(* CODESYS project Tutorial.export
   Author: ifm electronic
   Version: 3.4.0.0
   Description: Project template for 7" ifm ecomat display 64bit device
   Title: ifm_ecomatDisplay_64bit_7Inch
   CompiledLibraryCompatibilityVersion: CODESYS V3.5 SP16 Patch 5
   Company: ifm electronic

Project tree, tasks and I/O mapping:
  Device : ecomatDisplay_64bit, ifm electronic, version 3.5.19.78
    application Application
      libraries: Standard, 3.5.18.0 (System); ifm_ecomatDisplay_Cnt, * (ifm electronic)
      task Task (cyclic, interval t#10ms, priority 1) calls PLC_PRG, P_VehicleSpeed, P_DateTime, P_Main
      task VISU_TASK (cyclic, interval t#20ms, priority 15) calls VisuElems.Visu_Prg
      GlobalVariables/
        Enums/
          global variables ScreenIDs
        global variables GLV_MVC
        global variables GVL_KeyList
        global variables GVL_KeyList_FT
        global variables GVL_KeyList_RT
      MVC/
        Controller/
          MainScreen/
            function block FB_MainScreen [ST]
          Profiles/
          Settings/
            function block FB_Settings [ST]
          function block FB_Router [ST]
        Model/
          program P_DateTime [ST]
          program P_VehicleSpeed [ST]
        View/
          Settings/
            Widgets/
              visualisation Angle
              visualisation Graph
            visualisation Settings
          visualisation Background
          visualisation MainScreen
          visualisation Profiles
      TextLists/
        text list TL_eKeyMapCodes
      image pool ifmImagePool
      program PLC_PRG [FBD]: ACT_KeyList_FT, ACT_KeyList_RT
      program PLC_PRG_IN_ST [ST]: ACT_KeyList_FT, ACT_KeyList_RT
      program P_Main [ST]
    Communication : Communication, ifm electronic, version 3.5.19.78
      Ethernet : Ethernet, ifm electronic, version 3.5.19.78
      CAN : CAN, ifm electronic, version 3.5.19.78
        CANbus : CANbus, ifm electronic, version 3.0.0.0
          J1939_Manager : J1939_Manager, CODESYS, version 4.2.0.0
            RX_Tutorial : J1939_ECU, CODESYS, version 4.2.0.0
                settings: NAME = 16#0000000000000000; Communication Watchdog Timeout Period = 16#05DC ms; Activated PGs = 1; PG Offline Data.Name = "My_PGN"; PG Offline Data.Description = ""; PG Online Data.PGN = 65285; PG Online Data.Length (Bytes) = 8; PG Transmission Settings.Destination Address = 255; PG Transmission Settings.CycleTimeFactor = 1; Signal Offline Data.SPN = 1; Signal Offline Data.Name = "RX_Speed"; Signal Offline Data.Description = ""; Signal Offline Data.Unit = ""; Signal Offline Data.Min = 0; Signal Offline Data.Max = 0; Signal Online Data.BitSize = 8; Signal Online Data.BitPosition = 0; Convert Data.Flags = 3; Convert Data.pSigValue = 0; Convert Data.Scaling = 4607182418800017408; Convert Data.Offset = 0
                input  RX_Speed : USINT  // RX_Speed
            TX_Motor : J1939_ECU, CODESYS, version 4.2.0.0
                settings: NAME = 16#0000000000000000; Local Device = TRUE; Communication Watchdog Timeout Period = 16#05DC ms; Activated PGs = 1; PG Offline Data.Name = "TX_Speed"; PG Offline Data.Description = ""; PG Online Data.PGN = 65286; PG Online Data.Length (Bytes) = 8; PG Transmission Settings.Destination Address = 255; PG Transmission Settings.CycleTimeFactor = 5; Signal Offline Data.SPN = 0; Signal Offline Data.Name = "TX_ModifiedSpeed"; Signal Offline Data.Description = ""; Signal Offline Data.Unit = ""; Signal Offline Data.Min = 0; Signal Offline Data.Max = 0; Signal Online Data.BitSize = 8; Signal Online Data.BitPosition = 0; Convert Data.Flags = 3; Convert Data.pSigValue = 0; Convert Data.Scaling = 4607182418800017408; Convert Data.Offset = 0; Activated PGs = 0
                output Application.P_VehicleSpeed.uSpeed : USINT  // TX_ModifiedSpeed
  Project Information/
  text list GlobalTextList
  text list System
  5ce3da45-db07-42e7-a21c-a00fff4ed8f6|E:\BSR\Me\May Be Useful\ifm-engg_Logo\IFMLO_PANT_2c.png
  5ce3da45-db07-42e7-a21c-a00fff4ed8f6|E:\BSR\OnSVN\CODESYS_V3x\PDM360-3\DesignDocs\Pictures\7Inch\Bg_7Inch_dark.png
  5ce3da45-db07-42e7-a21c-a00fff4ed8f6|E:\BSR\OnSVN\CODESYS_V3x\PDM360-3\DesignDocs\Pictures\7Inch\Bg_7Inch_light.png
  5ce3da45-db07-42e7-a21c-a00fff4ed8f6|E:\BSR\OnSVN\CODESYS_V3x\PDM360-3\DesignDocs\Pictures\7Inch\Button_7Inch_dark.png
  5ce3da45-db07-42e7-a21c-a00fff4ed8f6|E:\BSR\OnSVN\CODESYS_V3x\PDM360-3\DesignDocs\Pictures\7Inch\Button_7Inch_light.png
  5ce3da45-db07-42e7-a21c-a00fff4ed8f6|E:\BSR\OnSVN\CODESYS_V3x\PDM360-3\DesignDocs\Pictures\7Inch\Button_And_Bg_7Inch_dark.png
  5ce3da45-db07-42e7-a21c-a00fff4ed8f6|E:\BSR\OnSVN\CODESYS_V3x\PDM360-3\DesignDocs\Pictures\7Inch\Button_And_Bg_7Inch_light.png
*)

// Device/Application/GlobalVariables/GLV_MVC

VAR_GLOBAL
	ScreenID : eScreenID := eScreenID.Main;
END_VAR

// Device/Application/GlobalVariables/GVL_KeyList
{attribute 'qualified_only'}

(* 

!!! This GVL list is from project template !!!

The following variables are controlled by key events mapped at Default Hotkey mapping list in Visualization Manager.

For example, F1 function key of standard keyboard (MFII) is pressed, xF1 bit in this list will become TRUE; when the same 
key is released then xF1 become FALSE.

*)

VAR_GLOBAL

(* Display system key press / release event status. TRUE = Key Pressed, FALSE = Key Released  *)
	xF1 		: BOOL;		(* Event status of F1 function key *)
	xF2 		: BOOL;		(* Event status of F2 function key *)
	xF3 		: BOOL;		(* Event status of F3 function key *)
	xF4 		: BOOL;		(* Event status of F4 function key *)
	xF5 		: BOOL;		(* Event status of F5 function key *)
	xF6 		: BOOL;		(* Event status of F6 function key *)
	xF7 		: BOOL;		(* Event status of F7 function key *)
	xF8 		: BOOL;		(* Event status of F8 function key *)
	xF9 		: BOOL;		(* Event status of F9 function key *)
	xF10 		: BOOL;		(* Event status of F10 function key *)
	xUp 		: BOOL;		(* Event status of Up arrow key *)
	xDown		: BOOL;		(* Event status of Down arrow key *)
	xLeft 		: BOOL;		(* Event status of Left arrow key *)
	xRight 		: BOOL;		(* Event status of Right arrow key *)
	xKey_Return : BOOL;		(* Event status of Return (or Enter) key *)
END_VAR

// Device/Application/GlobalVariables/GVL_KeyList_FT
{attribute 'qualified_only'}

(* 

!!! This GVL list is from project template !!!

The following variables returns a pulse for one scan cycle when a respective key is released (i.e. at falling trigger).
These key release event is detected by the state of variables in GVL GVL_KeyList.

For example, F1 function key of standard keyboard (MFII) is released, xF1 bit in this list will become TRUE for one scan cycle.

*)

VAR_GLOBAL

(* Display system key release event falling trigger pulse. *)
	xF1 		: BOOL;		(* Event status of F1 function key *)
	xF2 		: BOOL;		(* Event status of F2 function key *)
	xF3 		: BOOL;		(* Event status of F3 function key *)
	xF4 		: BOOL;		(* Event status of F4 function key *)
	xF5 		: BOOL;		(* Event status of F5 function key *)
	xF6 		: BOOL;		(* Event status of F6 function key *)
	xF7 		: BOOL;		(* Event status of F7 function key *)
	xF8 		: BOOL;		(* Event status of F8 function key *)
	xF9 		: BOOL;		(* Event status of F9 function key *)
	xF10 		: BOOL;		(* Event status of F10 function key *)
	xUp 		: BOOL;		(* Event status of Up arrow key *)
	xDown		: BOOL;		(* Event status of Down arrow key *)
	xLeft 		: BOOL;		(* Event status of Left arrow key *)
	xRight 		: BOOL;		(* Event status of Right arrow key *)
	xKey_Return : BOOL;		(* Event status of Return (or Enter) key *)
END_VAR

// Device/Application/GlobalVariables/GVL_KeyList_RT
{attribute 'qualified_only'}

(* 

!!! This GVL list is from project template !!!

The following variables returns a pulse for one scan cycle when a respective key is pressed (i.e. at rising trigger)
These key press event is detected by the state of variables in GVL GVL_KeyList.

For example, F1 function key of standard keyboard (MFII) is pressed, xF1 bit in this list will become TRUE for one scan cycle.

*)

VAR_GLOBAL

(*Display system key press event rising trigger pulse *)
	xF1 		: BOOL;		(* Event status of F1 function key *)
	xF2 		: BOOL;		(* Event status of F2 function key *)
	xF3 		: BOOL;		(* Event status of F3 function key *)
	xF4 		: BOOL;		(* Event status of F4 function key *)
	xF5 		: BOOL;		(* Event status of F5 function key *)
	xF6 		: BOOL;		(* Event status of F6 function key *)
	xF7 		: BOOL;		(* Event status of F7 function key *)
	xF8 		: BOOL;		(* Event status of F8 function key *)
	xF9 		: BOOL;		(* Event status of F9 function key *)
	xF10 		: BOOL;		(* Event status of F10 function key *)
	xUp 		: BOOL;		(* Event status of Up arrow key *)
	xDown		: BOOL;		(* Event status of Down arrow key *)
	xLeft 		: BOOL;		(* Event status of Left arrow key *)
	xRight 		: BOOL;		(* Event status of Right arrow key *)
	xKey_Return : BOOL;		(* Event status of Return (or Enter) key *)
END_VAR

// Device/Application/GlobalVariables/Enums/ScreenIDs
{attribute 'qualified_only'}
VAR_GLOBAL
END_VAR

TYPE eScreenID : (
  Main := 0,
  Settings := 1
);
END_TYPE

// Device/Application/PLC_PRG

(* !!! This POU is from project template !!! *)

PROGRAM PLC_PRG
VAR
(* Below is the FB instance with initial values to set default key mapping. The default key map is as per the default values set for ifmDevice.stKEY_MAP_LIST. *)
	fbSetKeyMapping		: ifmDevice.SetKeyMapping;

(* Below is the FB instance with initial values to hide splash screen and show CODESYS visualisation if a visualization exists in the application. In this case 
Visu_Default is displayed. *)
	fbHideSplashScreen	: ifmDevice.HideSplashScreen;

END_VAR
VAR // added by the converter: edge detectors and wires of the graphical bodies
    _ft1, _ft2, _ft3, _ft4, _ft5, _ft6, _ft7, _ft8, _ft9, _ft10, _ft11, _ft12, _ft13, _ft14, _ft15 : F_TRIG;
    _rt1, _rt2, _rt3, _rt4, _rt5, _rt6, _rt7, _rt8, _rt9, _rt10, _rt11, _rt12, _rt13, _rt14, _rt15 : R_TRIG;
END_VAR

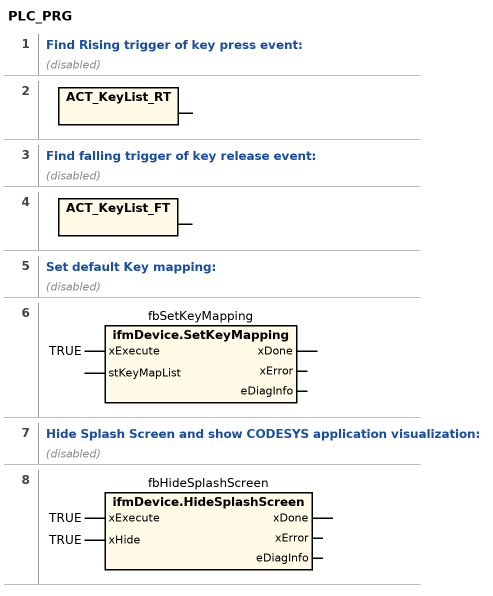
// NETWORK 1 (disabled)
// label: Find Rising trigger of key press event

// NETWORK 2
ACT_KeyList_RT();

// NETWORK 3 (disabled)
// label: Find falling trigger of key release event

// NETWORK 4
ACT_KeyList_FT();

// NETWORK 5 (disabled)
// label: Set default Key mapping

// NETWORK 6
fbSetKeyMapping(xExecute := TRUE); // ifmDevice.SetKeyMapping

// NETWORK 7 (disabled)
// label: Hide Splash Screen and show CODESYS application visualization

// NETWORK 8
fbHideSplashScreen(xExecute := TRUE, xHide := TRUE); // ifmDevice.HideSplashScreen

ACTION ACT_KeyList_FT:
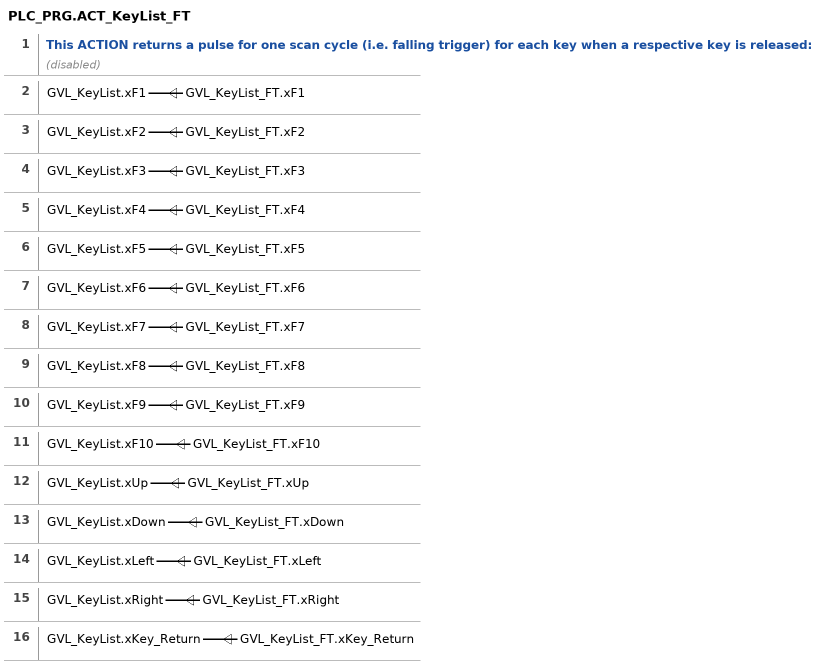
// NETWORK 1 (disabled)
// label: This ACTION returns a pulse for one scan cycle (i.e. falling trigger) for each key when a respective key is released

// NETWORK 2
_ft1(CLK := GVL_KeyList.xF1);
GVL_KeyList_FT.xF1 := _ft1.Q;

// NETWORK 3
_ft2(CLK := GVL_KeyList.xF2);
GVL_KeyList_FT.xF2 := _ft2.Q;

// NETWORK 4
_ft3(CLK := GVL_KeyList.xF3);
GVL_KeyList_FT.xF3 := _ft3.Q;

// NETWORK 5
_ft4(CLK := GVL_KeyList.xF4);
GVL_KeyList_FT.xF4 := _ft4.Q;

// NETWORK 6
_ft5(CLK := GVL_KeyList.xF5);
GVL_KeyList_FT.xF5 := _ft5.Q;

// NETWORK 7
_ft6(CLK := GVL_KeyList.xF6);
GVL_KeyList_FT.xF6 := _ft6.Q;

// NETWORK 8
_ft7(CLK := GVL_KeyList.xF7);
GVL_KeyList_FT.xF7 := _ft7.Q;

// NETWORK 9
_ft8(CLK := GVL_KeyList.xF8);
GVL_KeyList_FT.xF8 := _ft8.Q;

// NETWORK 10
_ft9(CLK := GVL_KeyList.xF9);
GVL_KeyList_FT.xF9 := _ft9.Q;

// NETWORK 11
_ft10(CLK := GVL_KeyList.xF10);
GVL_KeyList_FT.xF10 := _ft10.Q;

// NETWORK 12
_ft11(CLK := GVL_KeyList.xUp);
GVL_KeyList_FT.xUp := _ft11.Q;

// NETWORK 13
_ft12(CLK := GVL_KeyList.xDown);
GVL_KeyList_FT.xDown := _ft12.Q;

// NETWORK 14
_ft13(CLK := GVL_KeyList.xLeft);
GVL_KeyList_FT.xLeft := _ft13.Q;

// NETWORK 15
_ft14(CLK := GVL_KeyList.xRight);
GVL_KeyList_FT.xRight := _ft14.Q;

// NETWORK 16
_ft15(CLK := GVL_KeyList.xKey_Return);
GVL_KeyList_FT.xKey_Return := _ft15.Q;
END_ACTION

ACTION ACT_KeyList_RT:
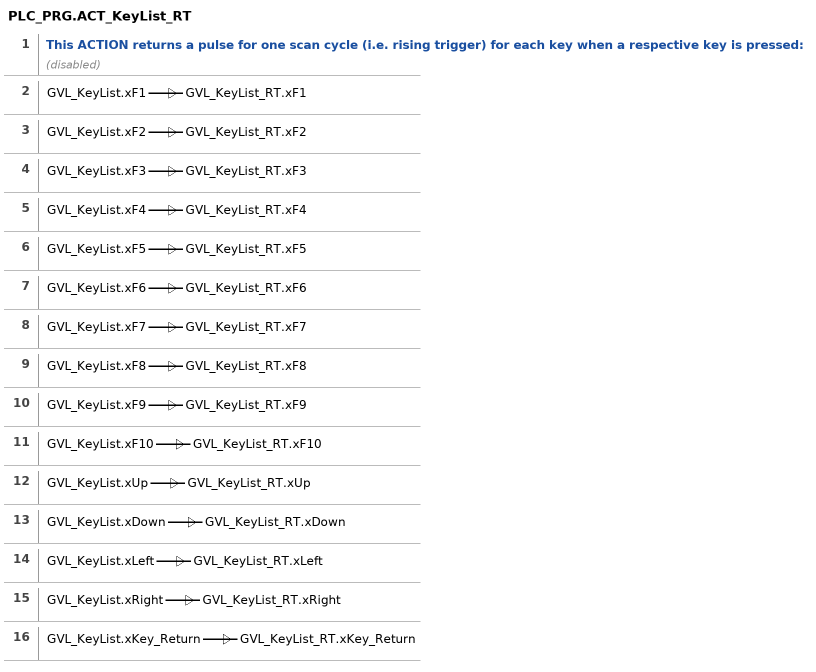
// NETWORK 1 (disabled)
// label: This ACTION returns a pulse for one scan cycle (i.e. rising trigger) for each key when a respective key is pressed

// NETWORK 2
_rt1(CLK := GVL_KeyList.xF1);
GVL_KeyList_RT.xF1 := _rt1.Q;

// NETWORK 3
_rt2(CLK := GVL_KeyList.xF2);
GVL_KeyList_RT.xF2 := _rt2.Q;

// NETWORK 4
_rt3(CLK := GVL_KeyList.xF3);
GVL_KeyList_RT.xF3 := _rt3.Q;

// NETWORK 5
_rt4(CLK := GVL_KeyList.xF4);
GVL_KeyList_RT.xF4 := _rt4.Q;

// NETWORK 6
_rt5(CLK := GVL_KeyList.xF5);
GVL_KeyList_RT.xF5 := _rt5.Q;

// NETWORK 7
_rt6(CLK := GVL_KeyList.xF6);
GVL_KeyList_RT.xF6 := _rt6.Q;

// NETWORK 8
_rt7(CLK := GVL_KeyList.xF7);
GVL_KeyList_RT.xF7 := _rt7.Q;

// NETWORK 9
_rt8(CLK := GVL_KeyList.xF8);
GVL_KeyList_RT.xF8 := _rt8.Q;

// NETWORK 10
_rt9(CLK := GVL_KeyList.xF9);
GVL_KeyList_RT.xF9 := _rt9.Q;

// NETWORK 11
_rt10(CLK := GVL_KeyList.xF10);
GVL_KeyList_RT.xF10 := _rt10.Q;

// NETWORK 12
_rt11(CLK := GVL_KeyList.xUp);
GVL_KeyList_RT.xUp := _rt11.Q;

// NETWORK 13
_rt12(CLK := GVL_KeyList.xDown);
GVL_KeyList_RT.xDown := _rt12.Q;

// NETWORK 14
_rt13(CLK := GVL_KeyList.xLeft);
GVL_KeyList_RT.xLeft := _rt13.Q;

// NETWORK 15
_rt14(CLK := GVL_KeyList.xRight);
GVL_KeyList_RT.xRight := _rt14.Q;

// NETWORK 16
_rt15(CLK := GVL_KeyList.xKey_Return);
GVL_KeyList_RT.xKey_Return := _rt15.Q;
END_ACTION

END_PROGRAM

// Device/Application/MVC/Model/P_VehicleSpeed
PROGRAM P_VehicleSpeed
VAR
	// currently requested speed
	uPercentage : USINT :=  0;
	
	// upper speed barier in km/h
	UPPER_SPEED_BARRIER : USINT := 190;
	
	// speed output for the motor
	uSpeed : USINT := 0;
END_VAR


// calculate our percentage from CAN input
uPercentage := RX_Speed * 10; 

// calculate the speed:  1% = 2km/h
IF (UPPER_SPEED_BARRIER < uPercentage * 2) THEN 	// check if the pedal is floored
	uSpeed := UPPER_SPEED_BARRIER; 					// if yes, allow only 95% of possible speed
	ELSE
	uSpeed := uPercentage * 2;					// else, use the calculated value
	
	
END_IF

END_PROGRAM

// Device/Application/MVC/Model/P_DateTime
PROGRAM P_DateTime
VAR
	GetSysTimeCyclic :ifmDevice.GetSysTime;
	DateTime :ifmDevice.stDATE_TIME;
END_VAR

GetSysTimeCyclic(
	xExecute:= TRUE , 
	xDone=> , 
	xError=> , 
	eDiagInfo=> , 
	stDateTime=> DateTime , 
	sTimeZone=> , 
	xNTP_DateTime=> );

END_PROGRAM

// Device/Application/P_Main
PROGRAM P_Main
VAR
	FB_Router : FB_Router;
END_VAR

FB_Router();

END_PROGRAM

// Device/Application/MVC/Controller/FB_Router
FUNCTION_BLOCK FB_Router
VAR_INPUT
END_VAR
VAR_OUTPUT
END_VAR
VAR
	FB_MainScreen : FB_MainScreen;
	FB_Settings : FB_Settings;
END_VAR




case ScreenID OF
		Main : FB_MainScreen();
		Settings : FB_Settings();
END_CASE

END_FUNCTION_BLOCK

// Device/Application/MVC/Controller/MainScreen/FB_MainScreen
FUNCTION_BLOCK FB_MainScreen
VAR_INPUT
END_VAR
VAR_OUTPUT
END_VAR
VAR
	uTest: udint := 0;
END_VAR

IF GVL_KeyList_FT.xF3 THEN
	ScreenID := 1;
END_IF

END_FUNCTION_BLOCK

// Device/Application/MVC/Controller/Settings/FB_Settings
FUNCTION_BLOCK FB_Settings
VAR_INPUT
END_VAR
VAR_OUTPUT
END_VAR
VAR
	MAX_WIDGET_INDEX :SINT := 1;
	// active widget index
	sWidgetIndex : SINT := 0;
END_VAR


// go back to HOME
IF GVL_KeyList_FT.xF5 THEN
	ScreenID := 0;
END_IF



// switch wigdet to left
IF GVL_KeyList_FT.xLeft THEN
    sWidgetIndex := (sWidgetIndex - 1 + MAX_WIDGET_INDEX + 1) MOD (MAX_WIDGET_INDEX + 1);
END_IF

// switch wigdet to right
IF GVL_KeyList_FT.xRight THEN
    sWidgetIndex := (sWidgetIndex + 1) MOD (MAX_WIDGET_INDEX + 1);
END_IF

END_FUNCTION_BLOCK

// Device/Application/PLC_PRG_IN_ST

(* !!! This POU is from project template !!! *)

PROGRAM PLC_PRG_IN_ST
VAR
(* Below is the FB instance with initial values to set default key mapping. The default key map is as per the default values set for ifmDevice.stKEY_MAP_LIST *)
	fbSetKeyMapping		: ifmDevice.SetKeyMapping;

(* Below is the FB instance with initial values to hide splash screen and show CODESYS visualisation if a visualization exists in the application. In this case 
Visu_Default is displayed. *)
	fbHideSplashScreen	: ifmDevice.HideSplashScreen;

(* Find rising trigger of key press event *)
	fbRTrig		: ARRAY[0..14] OF Standard.R_TRIG;
 
(* Find falling trigger of key release event *)
	fbFTrig		: ARRAY[0..14] OF Standard.F_TRIG; 
END_VAR

(* Find rising trigger of key press event *)
ACT_KeyList_RT();

(* Find falling trigger of key release event *)
ACT_KeyList_FT();


(* Set default key mapping *)
fbSetKeyMapping(
	xExecute		:= TRUE,
	stKeyMapList	:= , 
	xDone			=> , 
	xError			=> , 
	eDiagInfo		=> );

(* Hide splash screen and show CODESYS application visualization *)
fbHideSplashScreen(
	xExecute	:= TRUE,
	xHide		:= TRUE,
	xDone		=> , 
	xError		=> , 
	eDiagInfo	=> );

ACTION ACT_KeyList_FT:

(* This ACTION returns a pulse for one scan cycle (i.e. falling trigger) for each key when a respective key is released *)

fbFTrig[0](CLK := GVL_KeyList.xF1, 		Q => GVL_KeyList_FT.xF1);
fbFTrig[1](CLK := GVL_KeyList.xF2, 		Q => GVL_KeyList_FT.xF2);
fbFTrig[2](CLK := GVL_KeyList.xF3, 		Q => GVL_KeyList_FT.xF3);
fbFTrig[3](CLK := GVL_KeyList.xF4, 		Q => GVL_KeyList_FT.xF4);
fbFTrig[4](CLK := GVL_KeyList.xF5, 		Q => GVL_KeyList_FT.xF5);
fbFTrig[5](CLK := GVL_KeyList.xF6, 		Q => GVL_KeyList_FT.xF6);
fbFTrig[6](CLK := GVL_KeyList.xF7, 		Q => GVL_KeyList_FT.xF7);
fbFTrig[7](CLK := GVL_KeyList.xF8,		Q => GVL_KeyList_FT.xF8);
fbFTrig[8](CLK := GVL_KeyList.xF9, 		Q => GVL_KeyList_FT.xF9);
fbFTrig[9](CLK := GVL_KeyList.xF10, 	Q => GVL_KeyList_FT.xF10);

fbFTrig[10](CLK := GVL_KeyList.xUp, 	Q => GVL_KeyList_FT.xUp);
fbFTrig[11](CLK := GVL_KeyList.xDown,	Q => GVL_KeyList_FT.xDown);
fbFTrig[12](CLK := GVL_KeyList.xLeft,	Q => GVL_KeyList_FT.xLeft);
fbFTrig[13](CLK := GVL_KeyList.xRight,	Q => GVL_KeyList_FT.xRight);
fbFTrig[14](CLK := GVL_KeyList.xKey_Return, Q => GVL_KeyList_FT.xKey_Return);
END_ACTION

ACTION ACT_KeyList_RT:

(* This ACTION returns a pulse for one scan cycle (i.e. rising trigger) for each key when a respective key is pressed *)
fbRTrig[0](CLK := GVL_KeyList.xF1, 		Q => GVL_KeyList_RT.xF1);
fbRTrig[1](CLK := GVL_KeyList.xF2, 		Q => GVL_KeyList_RT.xF2);
fbRTrig[2](CLK := GVL_KeyList.xF3, 		Q => GVL_KeyList_RT.xF3);
fbRTrig[3](CLK := GVL_KeyList.xF4, 		Q => GVL_KeyList_RT.xF4);
fbRTrig[4](CLK := GVL_KeyList.xF5, 		Q => GVL_KeyList_RT.xF5);
fbRTrig[5](CLK := GVL_KeyList.xF6, 		Q => GVL_KeyList_RT.xF6);
fbRTrig[6](CLK := GVL_KeyList.xF7, 		Q => GVL_KeyList_RT.xF7);
fbRTrig[7](CLK := GVL_KeyList.xF8,		Q => GVL_KeyList_RT.xF8);
fbRTrig[8](CLK := GVL_KeyList.xF9, 		Q => GVL_KeyList_RT.xF9);
fbRTrig[9](CLK := GVL_KeyList.xF10, 	Q => GVL_KeyList_RT.xF10);

fbRTrig[10](CLK := GVL_KeyList.xUp, 	Q => GVL_KeyList_RT.xUp);
fbRTrig[11](CLK := GVL_KeyList.xDown,	Q => GVL_KeyList_RT.xDown);
fbRTrig[12](CLK := GVL_KeyList.xLeft,	Q => GVL_KeyList_RT.xLeft);
fbRTrig[13](CLK := GVL_KeyList.xRight,	Q => GVL_KeyList_RT.xRight);
fbRTrig[14](CLK := GVL_KeyList.xKey_Return, Q => GVL_KeyList_RT.xKey_Return);
END_ACTION

END_PROGRAM

// Device/Application/MVC/View/Background
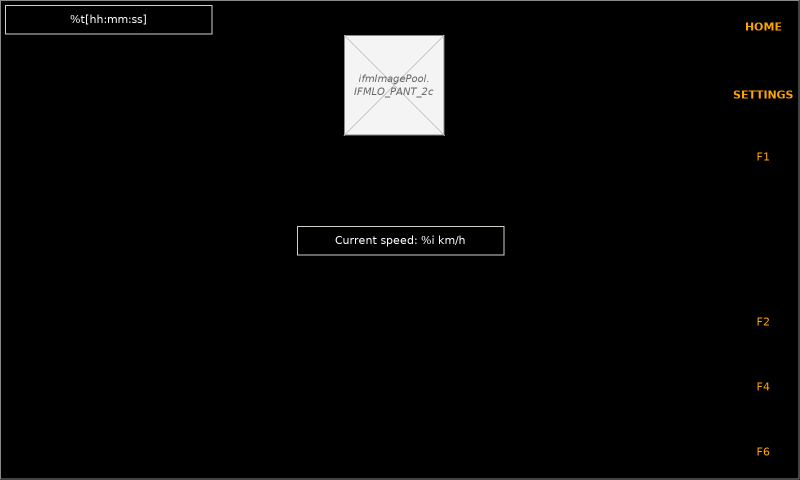
VISUALIZATION Background  // 800x480
    Frame (0,0 800x480), input disabled if: FALSE, frame switch variable: ScreenID
        shows MainScreen()
        shows Settings()
        shows Profiles()
END_VISUALIZATION

// Device/Application/MVC/View/MainScreen
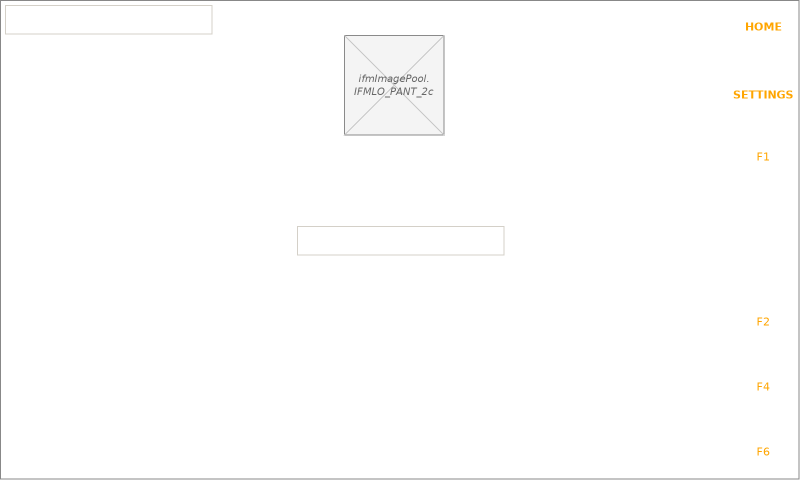
VISUALIZATION MainScreen  // 800x480, background image ifmImagePool.Button_And_Bg_7Inch_dark
    Rectangle (732,132 63x50), "F1"
    Rectangle (732,70 63x50), "SETTINGS"
    Rectangle (732,2 63x50), "HOME"
    Rectangle (732,297 63x50), "F2"
    Rectangle (732,362 63x50), "F4"
    Rectangle (732,427 63x50), "F6"
    Image (344,35 100x100), image: ifmImagePool.IFMLO_PANT_2c
    Textfield (5,5 207x29), "%t[hh:mm:ss]", text variable: P_DateTime.DateTime
    Textfield (297,226 207x29), "Current speed: %i km/h", text variable: P_VehicleSpeed.uSpeed
END_VISUALIZATION

// Device/Application/MVC/View/Profiles
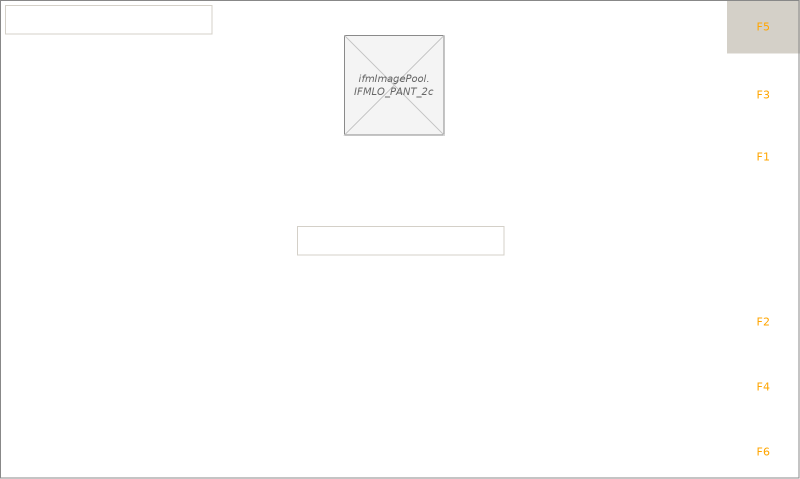
VISUALIZATION Profiles  // 800x479, background image ifmImagePool.Button_And_Bg_7Inch_dark
    Rectangle (727,-2 73x55), invisible if: not(ScreenID = eScreenID.Main)
    Rectangle (732,132 63x50), "F1"
    Rectangle (732,70 63x50), "F3"
    Rectangle (732,2 63x50), "F5"
    Rectangle (732,297 63x50), "F2"
    Rectangle (732,362 63x50), "F4"
    Rectangle (732,427 63x50), "F6"
    Image (344,35 100x100), image: ifmImagePool.IFMLO_PANT_2c
    Textfield (5,5 207x29), "%t[hh:mm:ss]", text variable: P_DateTime.DateTime
    Textfield (297,226 207x29), "Current speed: %i km/h", text variable: P_VehicleSpeed.uSpeed
END_VISUALIZATION

// Device/Application/MVC/View/Settings/Settings
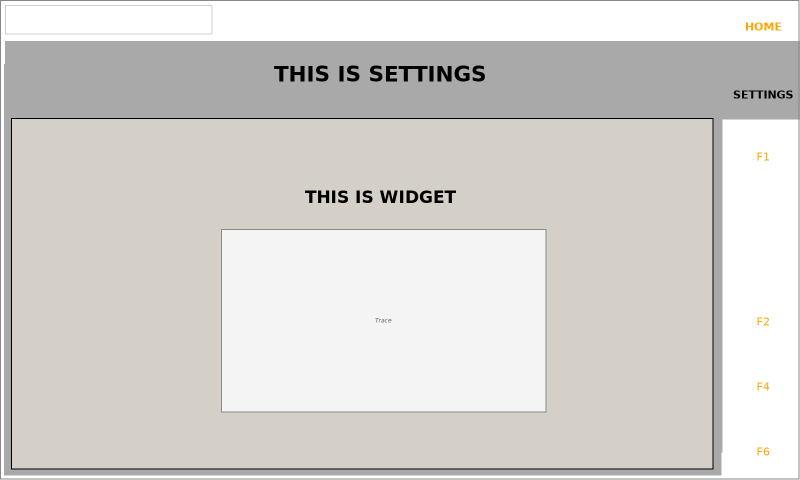
VISUALIZATION Settings  // 800x480, background image ifmImagePool.Button_And_Bg_7Inch_dark
    Group (4,41 796x434)
        Group (0,23 796x411)
            Rectangle (723,0 73x55)
            Rectangle (0,0 717x411)
            Rectangle (581,0 148x55)
        Group (1,0 717x421)
            Rectangle (723,0 73x55)
            Rectangle (0,0 717x411)
            Rectangle (581,0 148x55)
    Rectangle (732,132 63x50), "F1"
    Rectangle (732,70 63x50), "SETTINGS"
    Rectangle (732,2 63x50), "HOME"
    Rectangle (732,297 63x50), "F2"
    Rectangle (732,362 63x50), "F4"
    Rectangle (732,427 63x50), "F6"
    Textfield (5,5 207x29), "%t[hh:mm:ss]", text variable: P_DateTime.DateTime
    Rectangle (153,49 455x50), "THIS IS SETTINGS"
    Rectangle (11,118 702x351)
    Rectangle (153,172 455x50), "THIS IS WIDGET"
    Frame (221,229 325x183), frame switch variable: P_Main.FB_Router.FB_Settings.sWidgetIndex
        shows Graph()
        shows Angle()
END_VISUALIZATION

// Device/Application/MVC/View/Settings/Widgets/Angle
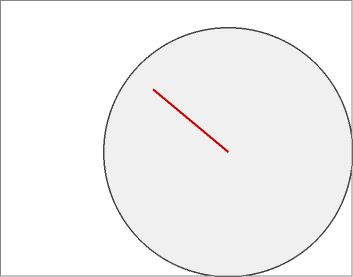
VISUALIZATION Angle  // 353x277
    Meter90 (103,27 250x250), value: P_VehicleSpeed.uSpeed, style: Meter-Meter90-Gray, scale format: %.1f, scale 0..100
END_VISUALIZATION

// Device/Application/MVC/View/Settings/Widgets/Graph
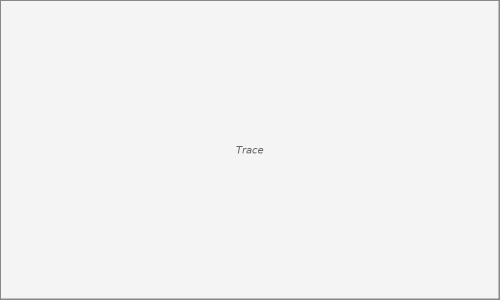
VISUALIZATION Graph  // 500x300
    Trace (0,0 500x300)
END_VISUALIZATION

(* text list System (id | default)
  Apr | Apr
  April | April
  Aug | Aug
  August | August
  Dec | Dec
  December | December
  Feb | Feb
  February | February
  Fri | Fri
  Friday | Friday
  Jan | Jan
  January | January
  Jul | Jul
  July | July
  Jun | Jun
  June | June
  Mar | Mar
  March | March
  May | May
  May_3Letter | May
  Mon | Mon
  Monday | Monday
  Nov | Nov
  November | November
  Oct | Oct
  October | October
  Sat | Sat
  Saturday | Saturday
  Sep | Sep
  September | September
  Sun | Sun
  Sunday | Sunday
  Thu | Thu
  Thursday | Thursday
  Tue | Tue
  Tuesday | Tuesday
  Wed | Wed
  Wednesday | Wednesday
   |  *)

(* text list TL_eKeyMapCodes (id | default)
  0 | NONE
  1 | ESCAPE
  74 | MINUS
  55 | ASTERISK
  57 | SPACE
  83 | COMMA
  98 | SLASH
  78 | PLUS
  11 | KEY_0
  2 | KEY_1
  3 | KEY_2
  4 | KEY_3
  5 | KEY_4
  6 | KEY_5
  7 | KEY_6
  8 | KEY_7
  9 | KEY_8
  10 | KEY_9
  30 | KEY_A
  48 | KEY_B
  46 | KEY_C
  32 | KEY_D
  18 | KEY_E
  33 | KEY_F
  34 | KEY_G
  35 | KEY_H
  23 | KEY_I
  36 | KEY_J
  37 | KEY_K
  38 | KEY_L
  50 | KEY_M
  49 | KEY_N
  24 | KEY_O
  25 | KEY_P
  16 | KEY_Q
  19 | KEY_R
  31 | KEY_S
  20 | KEY_T
  22 | KEY_U
  47 | KEY_V
  17 | KEY_W
  45 | KEY_X
  21 | KEY_Y
  44 | KEY_Z
  28 | KEY_RETURN
  14 | BACKSPACE
  15 | TAB
  99 | PRINT
  102 | HOME
  103 | UP
  105 | LEFT
  106 | RIGHT
  107 | END
  108 | DOWN
  110 | INSERT
  111 | DELETE
  119 | PAUSE
  59 | F1
  60 | F2
  61 | F3
  62 | F4
  63 | F5
  64 | F6
  65 | F7
  66 | F8
  67 | F9
  68 | F10
  87 | F11
  88 | F12
  82 | NUM0
  79 | NUM1
  80 | NUM2
  81 | NUM3
  75 | NUM4
  76 | NUM5
  77 | NUM6
  71 | NUM7
  72 | NUM8
  73 | NUM9
   |  *)
